// TIA Portal V17 export
// export: Created 2025-03-05T07:59:42.6499915Z, ExportSetting WithDefaults, DisplayName Totally Integrated Automation Portal, DisplayVersion V17 Update 8, DisplayName TIA Portal Openness, DisplayVersion V17 Update 8, DisplayName TIA Portal Version Control Interface, DisplayVersion V17, DisplayName SINAMICS Startdrive Advanced, DisplayVersion V17 SP2, DisplayName SINAMICS Startdrive G110M, G120, G120C, G120D, G120P, G115D, DisplayVersion V17 SP2, DisplayName SINAMICS Startdrive G130, G150, S120, S150, SINAMICS MV, S210, DisplayVersion V17 SP2, DisplayName STEP 7 Professional, DisplayVersion V17 Update 8, DisplayName SINUMERIK ONE STEP 7 Toolbox, DisplayVersion V17 Update 12, DisplayName SINUMERIK 840D sl STEP 7 Toolbox, DisplayVersion V17 Update 12, DisplayName STEP 7 Safety, DisplayVersion V17 Update 6, DisplayName WinCC Advanced, DisplayVersion V17 Update 8
FUNCTION "FC361_NCK_M_CH5_UNIT_2_STA_2" : Void   // FC361, LAD
TITLE = Channel 1 data
{ S7_Optimized_Access := 'FALSE' }
AUTHOR : ETXETAR
VERSION : 1.0
// stored: AutoNumber false, IsIECCheckEnabled false, SetENOAutomatically false, UDAEnableTagReadback false
BEGIN

REGION Network 1: ACKNOWLEDGE M700-FIXTURE 4 CLAMP SEQUENCE (READ-IN DISABLE) / ACKNOWLEDGE M100-CLAMP SEQUENCE FIXTURE 1
   // NOTE: WHEN THERE IS NOT INDEXING TABLE AVAILABLE IN THE MACHINE DELETE 
   // DB2171.DBX5.0 AND DB2171.DBX2.0
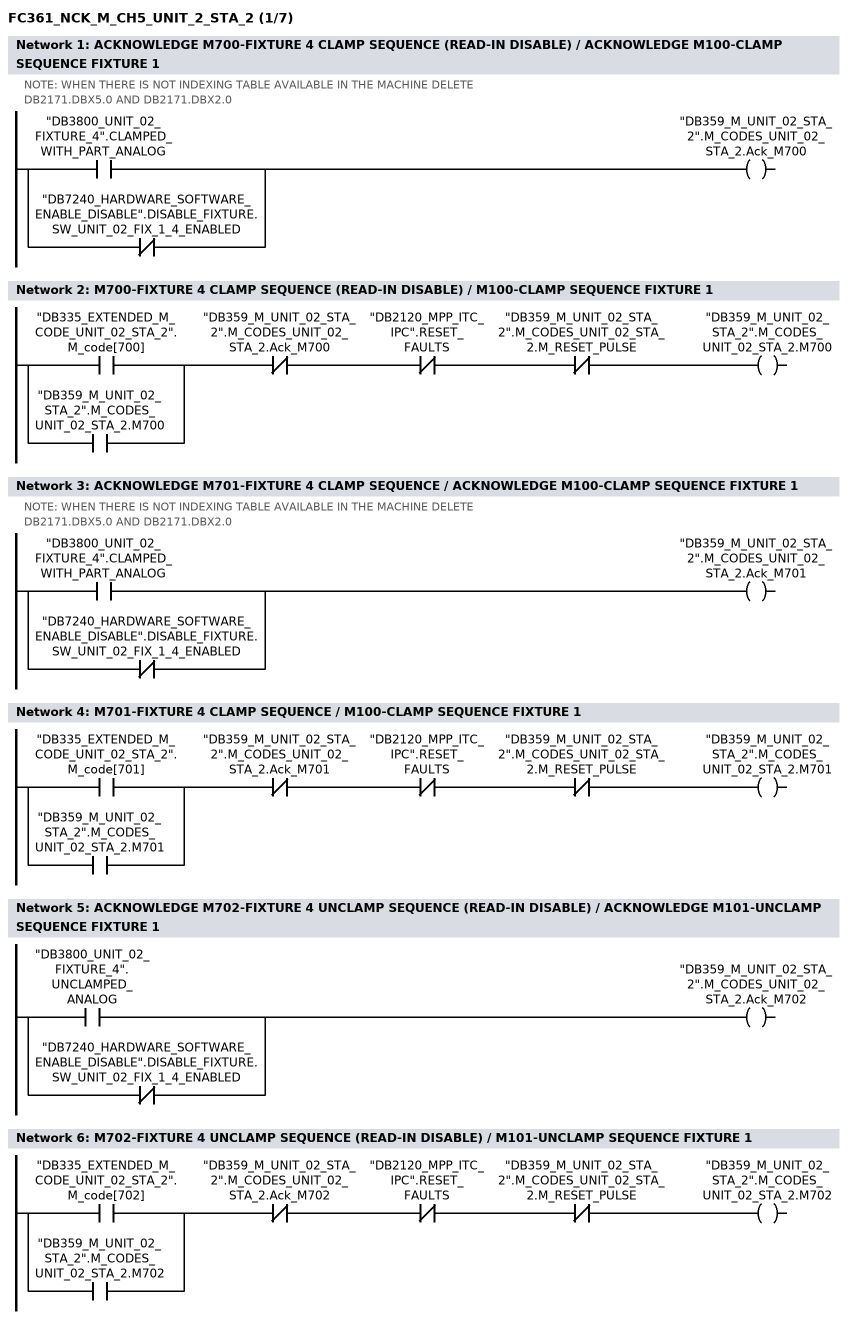
   RUNG wire#powerrail
      Contact( "DB3800_UNIT_02_FIXTURE_4".CLAMPED_WITH_PART_ANALOG )
      wire#w1
      Coil( "DB359_M_UNIT_02_STA_2".M_CODES_UNIT_02_STA_2.Ack_M700 )
   END_RUNG
   RUNG wire#powerrail
      I_Contact( "DB7240_HARDWARE_SOFTWARE_ENABLE_DISABLE".DISABLE_FIXTURE.SW_UNIT_02_FIX_1_4_ENABLED )
   END_RUNG wire#w1
   // the same network as SCL:
   "DB359_M_UNIT_02_STA_2".M_CODES_UNIT_02_STA_2.Ack_M700 := "DB3800_UNIT_02_FIXTURE_4".CLAMPED_WITH_PART_ANALOG OR NOT "DB7240_HARDWARE_SOFTWARE_ENABLE_DISABLE".DISABLE_FIXTURE.SW_UNIT_02_FIX_1_4_ENABLED;
END_REGION

REGION Network 2: M700-FIXTURE 4 CLAMP SEQUENCE (READ-IN DISABLE) / M100-CLAMP SEQUENCE FIXTURE 1
   RUNG wire#powerrail
      Contact( "DB335_EXTENDED_M_CODE_UNIT_02_STA_2".M_code[700] )
      wire#w1
      I_Contact( "DB359_M_UNIT_02_STA_2".M_CODES_UNIT_02_STA_2.Ack_M700 )
      I_Contact( "DB2120_MPP_ITC_IPC".RESET_FAULTS )
      I_Contact( "DB359_M_UNIT_02_STA_2".M_CODES_UNIT_02_STA_2.M_RESET_PULSE )
      Coil( "DB359_M_UNIT_02_STA_2".M_CODES_UNIT_02_STA_2.M700 )
   END_RUNG
   RUNG wire#powerrail
      Contact( "DB359_M_UNIT_02_STA_2".M_CODES_UNIT_02_STA_2.M700 )
   END_RUNG wire#w1
   // the same network as SCL:
   "DB359_M_UNIT_02_STA_2".M_CODES_UNIT_02_STA_2.M700 := ("DB335_EXTENDED_M_CODE_UNIT_02_STA_2".M_code[700] OR "DB359_M_UNIT_02_STA_2".M_CODES_UNIT_02_STA_2.M700) AND NOT "DB359_M_UNIT_02_STA_2".M_CODES_UNIT_02_STA_2.Ack_M700 AND NOT "DB2120_MPP_ITC_IPC".RESET_FAULTS AND NOT "DB359_M_UNIT_02_STA_2".M_CODES_UNIT_02_STA_2.M_RESET_PULSE;
END_REGION

REGION Network 3: ACKNOWLEDGE M701-FIXTURE 4 CLAMP SEQUENCE / ACKNOWLEDGE M100-CLAMP SEQUENCE FIXTURE 1
   // NOTE: WHEN THERE IS NOT INDEXING TABLE AVAILABLE IN THE MACHINE DELETE 
   // DB2171.DBX5.0 AND DB2171.DBX2.0
   RUNG wire#powerrail
      Contact( "DB3800_UNIT_02_FIXTURE_4".CLAMPED_WITH_PART_ANALOG )
      wire#w1
      Coil( "DB359_M_UNIT_02_STA_2".M_CODES_UNIT_02_STA_2.Ack_M701 )
   END_RUNG
   RUNG wire#powerrail
      I_Contact( "DB7240_HARDWARE_SOFTWARE_ENABLE_DISABLE".DISABLE_FIXTURE.SW_UNIT_02_FIX_1_4_ENABLED )
   END_RUNG wire#w1
   // the same network as SCL:
   "DB359_M_UNIT_02_STA_2".M_CODES_UNIT_02_STA_2.Ack_M701 := "DB3800_UNIT_02_FIXTURE_4".CLAMPED_WITH_PART_ANALOG OR NOT "DB7240_HARDWARE_SOFTWARE_ENABLE_DISABLE".DISABLE_FIXTURE.SW_UNIT_02_FIX_1_4_ENABLED;
END_REGION

REGION Network 4: M701-FIXTURE 4 CLAMP SEQUENCE / M100-CLAMP SEQUENCE FIXTURE 1
   RUNG wire#powerrail
      Contact( "DB335_EXTENDED_M_CODE_UNIT_02_STA_2".M_code[701] )
      wire#w1
      I_Contact( "DB359_M_UNIT_02_STA_2".M_CODES_UNIT_02_STA_2.Ack_M701 )
      I_Contact( "DB2120_MPP_ITC_IPC".RESET_FAULTS )
      I_Contact( "DB359_M_UNIT_02_STA_2".M_CODES_UNIT_02_STA_2.M_RESET_PULSE )
      Coil( "DB359_M_UNIT_02_STA_2".M_CODES_UNIT_02_STA_2.M701 )
   END_RUNG
   RUNG wire#powerrail
      Contact( "DB359_M_UNIT_02_STA_2".M_CODES_UNIT_02_STA_2.M701 )
   END_RUNG wire#w1
   // the same network as SCL:
   "DB359_M_UNIT_02_STA_2".M_CODES_UNIT_02_STA_2.M701 := ("DB335_EXTENDED_M_CODE_UNIT_02_STA_2".M_code[701] OR "DB359_M_UNIT_02_STA_2".M_CODES_UNIT_02_STA_2.M701) AND NOT "DB359_M_UNIT_02_STA_2".M_CODES_UNIT_02_STA_2.Ack_M701 AND NOT "DB2120_MPP_ITC_IPC".RESET_FAULTS AND NOT "DB359_M_UNIT_02_STA_2".M_CODES_UNIT_02_STA_2.M_RESET_PULSE;
END_REGION

REGION Network 5: ACKNOWLEDGE M702-FIXTURE 4 UNCLAMP SEQUENCE (READ-IN DISABLE) / ACKNOWLEDGE M101-UNCLAMP SEQUENCE FIXTURE 1
   RUNG wire#powerrail
      Contact( "DB3800_UNIT_02_FIXTURE_4".UNCLAMPED_ANALOG )
      wire#w1
      Coil( "DB359_M_UNIT_02_STA_2".M_CODES_UNIT_02_STA_2.Ack_M702 )
   END_RUNG
   RUNG wire#powerrail
      I_Contact( "DB7240_HARDWARE_SOFTWARE_ENABLE_DISABLE".DISABLE_FIXTURE.SW_UNIT_02_FIX_1_4_ENABLED )
   END_RUNG wire#w1
   // the same network as SCL:
   "DB359_M_UNIT_02_STA_2".M_CODES_UNIT_02_STA_2.Ack_M702 := "DB3800_UNIT_02_FIXTURE_4".UNCLAMPED_ANALOG OR NOT "DB7240_HARDWARE_SOFTWARE_ENABLE_DISABLE".DISABLE_FIXTURE.SW_UNIT_02_FIX_1_4_ENABLED;
END_REGION

REGION Network 6: M702-FIXTURE 4 UNCLAMP SEQUENCE (READ-IN DISABLE) / M101-UNCLAMP SEQUENCE FIXTURE 1
   RUNG wire#powerrail
      Contact( "DB335_EXTENDED_M_CODE_UNIT_02_STA_2".M_code[702] )
      wire#w1
      I_Contact( "DB359_M_UNIT_02_STA_2".M_CODES_UNIT_02_STA_2.Ack_M702 )
      I_Contact( "DB2120_MPP_ITC_IPC".RESET_FAULTS )
      I_Contact( "DB359_M_UNIT_02_STA_2".M_CODES_UNIT_02_STA_2.M_RESET_PULSE )
      Coil( "DB359_M_UNIT_02_STA_2".M_CODES_UNIT_02_STA_2.M702 )
   END_RUNG
   RUNG wire#powerrail
      Contact( "DB359_M_UNIT_02_STA_2".M_CODES_UNIT_02_STA_2.M702 )
   END_RUNG wire#w1
   // the same network as SCL:
   "DB359_M_UNIT_02_STA_2".M_CODES_UNIT_02_STA_2.M702 := ("DB335_EXTENDED_M_CODE_UNIT_02_STA_2".M_code[702] OR "DB359_M_UNIT_02_STA_2".M_CODES_UNIT_02_STA_2.M702) AND NOT "DB359_M_UNIT_02_STA_2".M_CODES_UNIT_02_STA_2.Ack_M702 AND NOT "DB2120_MPP_ITC_IPC".RESET_FAULTS AND NOT "DB359_M_UNIT_02_STA_2".M_CODES_UNIT_02_STA_2.M_RESET_PULSE;
END_REGION

REGION Network 7: ACKNOWLEDGE M703-FIXTURE 4 UNCLAMP SEQUENCE / ACKNOWLEDGE M101-UNCLAMP SEQUENCE FIXTURE 1
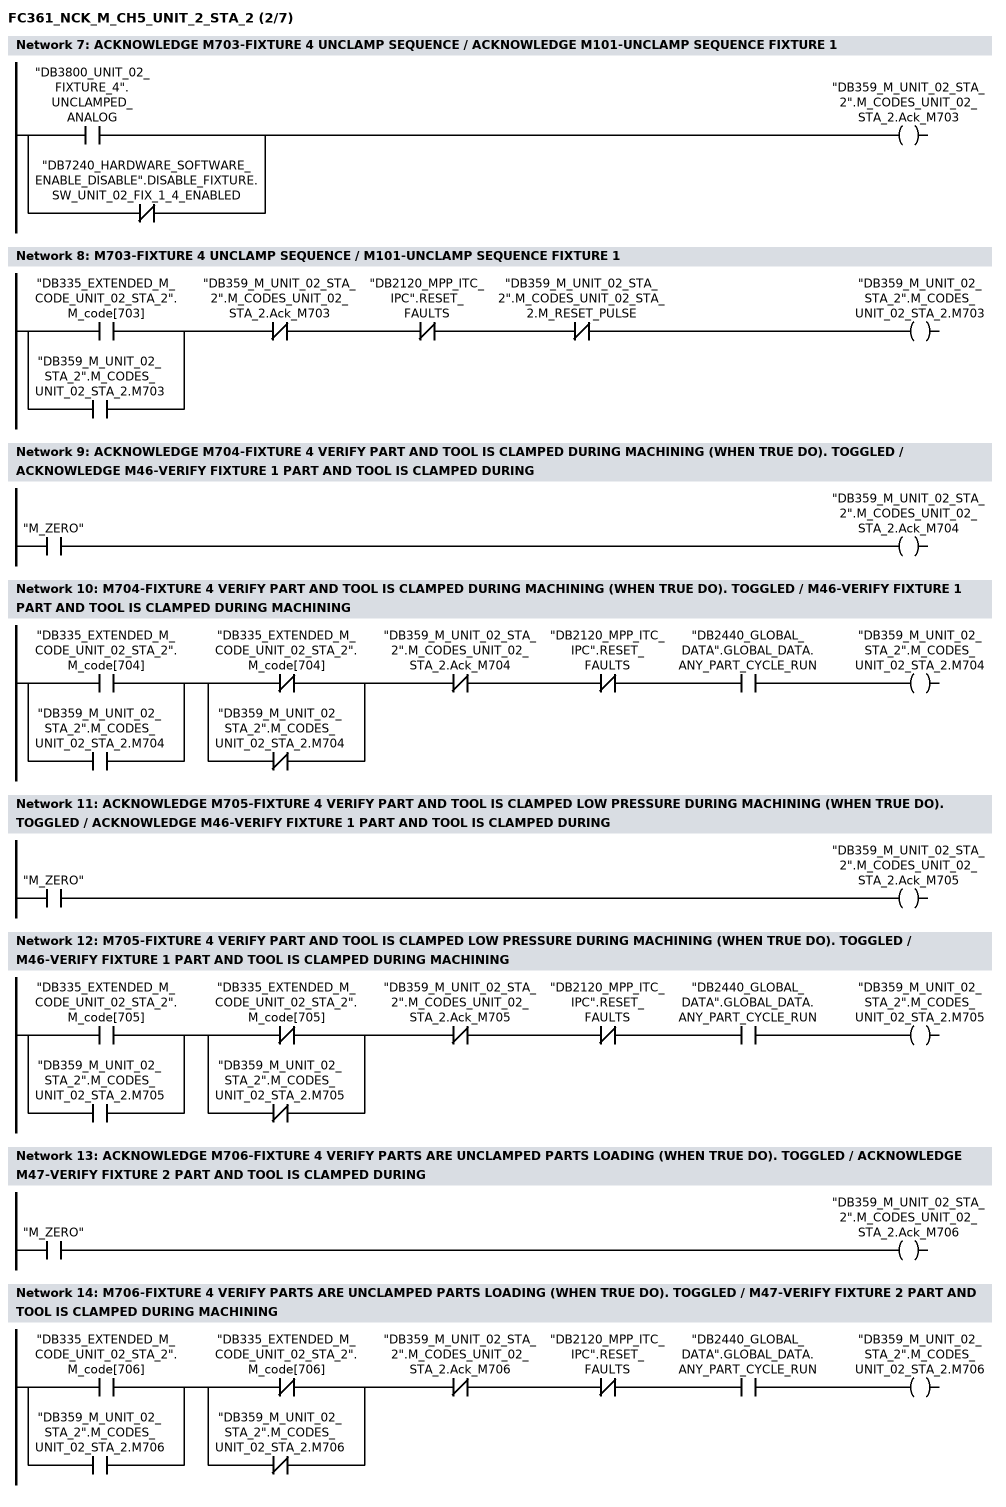
   RUNG wire#powerrail
      Contact( "DB3800_UNIT_02_FIXTURE_4".UNCLAMPED_ANALOG )
      wire#w1
      Coil( "DB359_M_UNIT_02_STA_2".M_CODES_UNIT_02_STA_2.Ack_M703 )
   END_RUNG
   RUNG wire#powerrail
      I_Contact( "DB7240_HARDWARE_SOFTWARE_ENABLE_DISABLE".DISABLE_FIXTURE.SW_UNIT_02_FIX_1_4_ENABLED )
   END_RUNG wire#w1
   // the same network as SCL:
   "DB359_M_UNIT_02_STA_2".M_CODES_UNIT_02_STA_2.Ack_M703 := "DB3800_UNIT_02_FIXTURE_4".UNCLAMPED_ANALOG OR NOT "DB7240_HARDWARE_SOFTWARE_ENABLE_DISABLE".DISABLE_FIXTURE.SW_UNIT_02_FIX_1_4_ENABLED;
END_REGION

REGION Network 8: M703-FIXTURE 4 UNCLAMP SEQUENCE / M101-UNCLAMP SEQUENCE FIXTURE 1
   RUNG wire#powerrail
      Contact( "DB335_EXTENDED_M_CODE_UNIT_02_STA_2".M_code[703] )
      wire#w1
      I_Contact( "DB359_M_UNIT_02_STA_2".M_CODES_UNIT_02_STA_2.Ack_M703 )
      I_Contact( "DB2120_MPP_ITC_IPC".RESET_FAULTS )
      I_Contact( "DB359_M_UNIT_02_STA_2".M_CODES_UNIT_02_STA_2.M_RESET_PULSE )
      Coil( "DB359_M_UNIT_02_STA_2".M_CODES_UNIT_02_STA_2.M703 )
   END_RUNG
   RUNG wire#powerrail
      Contact( "DB359_M_UNIT_02_STA_2".M_CODES_UNIT_02_STA_2.M703 )
   END_RUNG wire#w1
   // the same network as SCL:
   "DB359_M_UNIT_02_STA_2".M_CODES_UNIT_02_STA_2.M703 := ("DB335_EXTENDED_M_CODE_UNIT_02_STA_2".M_code[703] OR "DB359_M_UNIT_02_STA_2".M_CODES_UNIT_02_STA_2.M703) AND NOT "DB359_M_UNIT_02_STA_2".M_CODES_UNIT_02_STA_2.Ack_M703 AND NOT "DB2120_MPP_ITC_IPC".RESET_FAULTS AND NOT "DB359_M_UNIT_02_STA_2".M_CODES_UNIT_02_STA_2.M_RESET_PULSE;
END_REGION

REGION Network 9: ACKNOWLEDGE M704-FIXTURE 4 VERIFY PART AND TOOL IS CLAMPED DURING MACHINING (WHEN TRUE DO). TOGGLED / ACKNOWLEDGE M46-VERIFY FIXTURE 1 PART AND TOOL IS CLAMPED DURING
   RUNG wire#powerrail
      Contact( "M_ZERO" )
      Coil( "DB359_M_UNIT_02_STA_2".M_CODES_UNIT_02_STA_2.Ack_M704 )
   END_RUNG
   // the same network as SCL:
   "DB359_M_UNIT_02_STA_2".M_CODES_UNIT_02_STA_2.Ack_M704 := "M_ZERO";
END_REGION

REGION Network 10: M704-FIXTURE 4 VERIFY PART AND TOOL IS CLAMPED DURING MACHINING (WHEN TRUE DO). TOGGLED / M46-VERIFY FIXTURE 1 PART AND TOOL IS CLAMPED DURING MACHINING
   RUNG wire#powerrail
      Contact( "DB335_EXTENDED_M_CODE_UNIT_02_STA_2".M_code[704] )
      wire#w1
      I_Contact( "DB335_EXTENDED_M_CODE_UNIT_02_STA_2".M_code[704] )
      wire#w2
      I_Contact( "DB359_M_UNIT_02_STA_2".M_CODES_UNIT_02_STA_2.Ack_M704 )
      I_Contact( "DB2120_MPP_ITC_IPC".RESET_FAULTS )
      Contact( "DB2440_GLOBAL_DATA".GLOBAL_DATA.ANY_PART_CYCLE_RUN )
      Coil( "DB359_M_UNIT_02_STA_2".M_CODES_UNIT_02_STA_2.M704 )
   END_RUNG
   RUNG wire#powerrail
      Contact( "DB359_M_UNIT_02_STA_2".M_CODES_UNIT_02_STA_2.M704 )
   END_RUNG wire#w1
   RUNG wire#w1
      I_Contact( "DB359_M_UNIT_02_STA_2".M_CODES_UNIT_02_STA_2.M704 )
   END_RUNG wire#w2
   // the same network as SCL:
   "DB359_M_UNIT_02_STA_2".M_CODES_UNIT_02_STA_2.M704 := ("DB335_EXTENDED_M_CODE_UNIT_02_STA_2".M_code[704] OR "DB359_M_UNIT_02_STA_2".M_CODES_UNIT_02_STA_2.M704) AND (NOT "DB335_EXTENDED_M_CODE_UNIT_02_STA_2".M_code[704] OR NOT "DB359_M_UNIT_02_STA_2".M_CODES_UNIT_02_STA_2.M704) AND NOT "DB359_M_UNIT_02_STA_2".M_CODES_UNIT_02_STA_2.Ack_M704 AND NOT "DB2120_MPP_ITC_IPC".RESET_FAULTS AND "DB2440_GLOBAL_DATA".GLOBAL_DATA.ANY_PART_CYCLE_RUN;
END_REGION

REGION Network 11: ACKNOWLEDGE M705-FIXTURE 4 VERIFY PART AND TOOL IS CLAMPED LOW PRESSURE DURING MACHINING (WHEN TRUE DO). TOGGLED / ACKNOWLEDGE M46-VERIFY FIXTURE 1 PART AND TOOL IS CLAMPED DURING
   RUNG wire#powerrail
      Contact( "M_ZERO" )
      Coil( "DB359_M_UNIT_02_STA_2".M_CODES_UNIT_02_STA_2.Ack_M705 )
   END_RUNG
   // the same network as SCL:
   "DB359_M_UNIT_02_STA_2".M_CODES_UNIT_02_STA_2.Ack_M705 := "M_ZERO";
END_REGION

REGION Network 12: M705-FIXTURE 4 VERIFY PART AND TOOL IS CLAMPED LOW PRESSURE DURING MACHINING (WHEN TRUE DO). TOGGLED / M46-VERIFY FIXTURE 1 PART AND TOOL IS CLAMPED DURING MACHINING
   RUNG wire#powerrail
      Contact( "DB335_EXTENDED_M_CODE_UNIT_02_STA_2".M_code[705] )
      wire#w1
      I_Contact( "DB335_EXTENDED_M_CODE_UNIT_02_STA_2".M_code[705] )
      wire#w2
      I_Contact( "DB359_M_UNIT_02_STA_2".M_CODES_UNIT_02_STA_2.Ack_M705 )
      I_Contact( "DB2120_MPP_ITC_IPC".RESET_FAULTS )
      Contact( "DB2440_GLOBAL_DATA".GLOBAL_DATA.ANY_PART_CYCLE_RUN )
      Coil( "DB359_M_UNIT_02_STA_2".M_CODES_UNIT_02_STA_2.M705 )
   END_RUNG
   RUNG wire#powerrail
      Contact( "DB359_M_UNIT_02_STA_2".M_CODES_UNIT_02_STA_2.M705 )
   END_RUNG wire#w1
   RUNG wire#w1
      I_Contact( "DB359_M_UNIT_02_STA_2".M_CODES_UNIT_02_STA_2.M705 )
   END_RUNG wire#w2
   // the same network as SCL:
   "DB359_M_UNIT_02_STA_2".M_CODES_UNIT_02_STA_2.M705 := ("DB335_EXTENDED_M_CODE_UNIT_02_STA_2".M_code[705] OR "DB359_M_UNIT_02_STA_2".M_CODES_UNIT_02_STA_2.M705) AND (NOT "DB335_EXTENDED_M_CODE_UNIT_02_STA_2".M_code[705] OR NOT "DB359_M_UNIT_02_STA_2".M_CODES_UNIT_02_STA_2.M705) AND NOT "DB359_M_UNIT_02_STA_2".M_CODES_UNIT_02_STA_2.Ack_M705 AND NOT "DB2120_MPP_ITC_IPC".RESET_FAULTS AND "DB2440_GLOBAL_DATA".GLOBAL_DATA.ANY_PART_CYCLE_RUN;
END_REGION

REGION Network 13: ACKNOWLEDGE M706-FIXTURE 4 VERIFY PARTS ARE UNCLAMPED PARTS LOADING (WHEN TRUE DO). TOGGLED / ACKNOWLEDGE M47-VERIFY FIXTURE 2 PART AND TOOL IS CLAMPED DURING
   RUNG wire#powerrail
      Contact( "M_ZERO" )
      Coil( "DB359_M_UNIT_02_STA_2".M_CODES_UNIT_02_STA_2.Ack_M706 )
   END_RUNG
   // the same network as SCL:
   "DB359_M_UNIT_02_STA_2".M_CODES_UNIT_02_STA_2.Ack_M706 := "M_ZERO";
END_REGION

REGION Network 14: M706-FIXTURE 4 VERIFY PARTS ARE UNCLAMPED PARTS LOADING (WHEN TRUE DO). TOGGLED / M47-VERIFY FIXTURE 2 PART AND TOOL IS CLAMPED DURING MACHINING
   RUNG wire#powerrail
      Contact( "DB335_EXTENDED_M_CODE_UNIT_02_STA_2".M_code[706] )
      wire#w1
      I_Contact( "DB335_EXTENDED_M_CODE_UNIT_02_STA_2".M_code[706] )
      wire#w2
      I_Contact( "DB359_M_UNIT_02_STA_2".M_CODES_UNIT_02_STA_2.Ack_M706 )
      I_Contact( "DB2120_MPP_ITC_IPC".RESET_FAULTS )
      Contact( "DB2440_GLOBAL_DATA".GLOBAL_DATA.ANY_PART_CYCLE_RUN )
      Coil( "DB359_M_UNIT_02_STA_2".M_CODES_UNIT_02_STA_2.M706 )
   END_RUNG
   RUNG wire#powerrail
      Contact( "DB359_M_UNIT_02_STA_2".M_CODES_UNIT_02_STA_2.M706 )
   END_RUNG wire#w1
   RUNG wire#w1
      I_Contact( "DB359_M_UNIT_02_STA_2".M_CODES_UNIT_02_STA_2.M706 )
   END_RUNG wire#w2
   // the same network as SCL:
   "DB359_M_UNIT_02_STA_2".M_CODES_UNIT_02_STA_2.M706 := ("DB335_EXTENDED_M_CODE_UNIT_02_STA_2".M_code[706] OR "DB359_M_UNIT_02_STA_2".M_CODES_UNIT_02_STA_2.M706) AND (NOT "DB335_EXTENDED_M_CODE_UNIT_02_STA_2".M_code[706] OR NOT "DB359_M_UNIT_02_STA_2".M_CODES_UNIT_02_STA_2.M706) AND NOT "DB359_M_UNIT_02_STA_2".M_CODES_UNIT_02_STA_2.Ack_M706 AND NOT "DB2120_MPP_ITC_IPC".RESET_FAULTS AND "DB2440_GLOBAL_DATA".GLOBAL_DATA.ANY_PART_CYCLE_RUN;
END_REGION

REGION Network 15: ACKNOWLEDGE M707-FIXTURE 4 VERIFY FIXTURE REMAINS CLAMPED
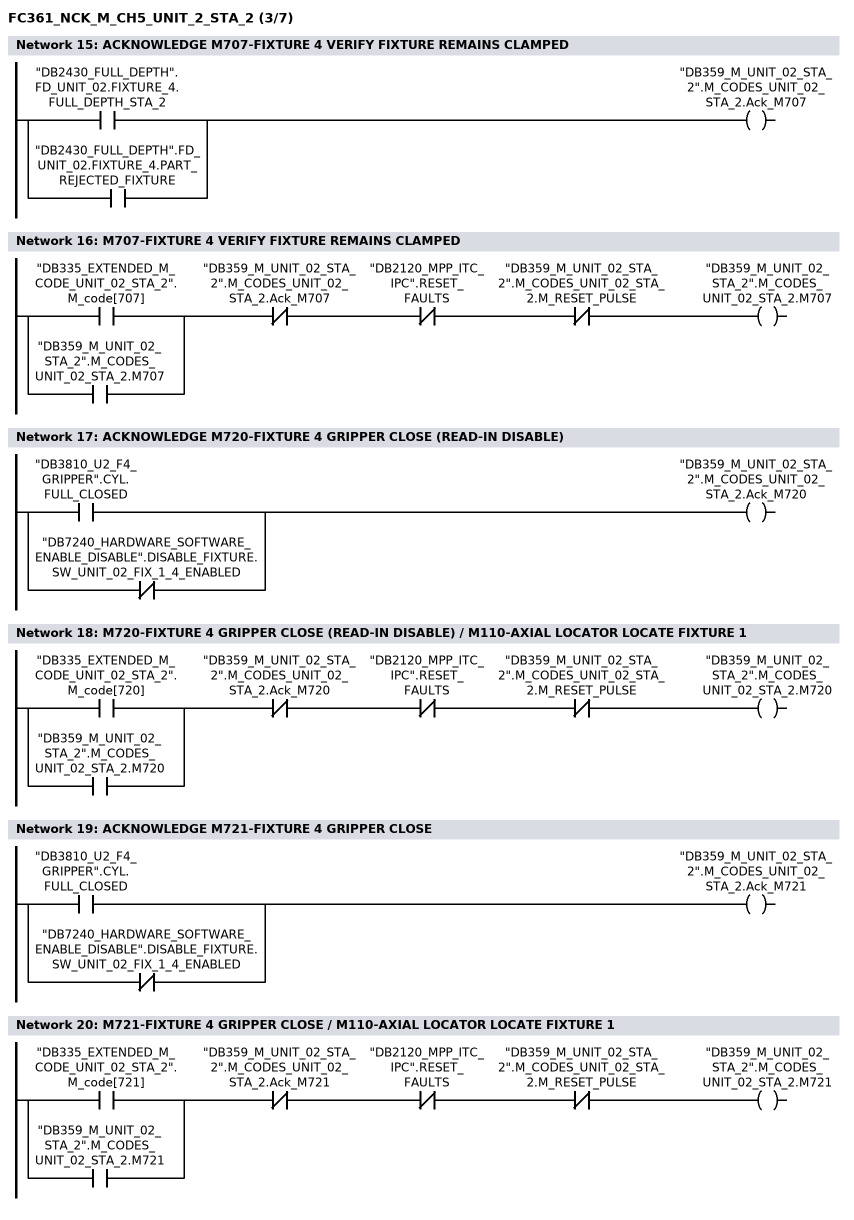
   RUNG wire#powerrail
      Contact( "DB2430_FULL_DEPTH".FD_UNIT_02.FIXTURE_4.FULL_DEPTH_STA_2 )
      wire#w1
      Coil( "DB359_M_UNIT_02_STA_2".M_CODES_UNIT_02_STA_2.Ack_M707 )
   END_RUNG
   RUNG wire#powerrail
      Contact( "DB2430_FULL_DEPTH".FD_UNIT_02.FIXTURE_4.PART_REJECTED_FIXTURE )
   END_RUNG wire#w1
   // the same network as SCL:
   "DB359_M_UNIT_02_STA_2".M_CODES_UNIT_02_STA_2.Ack_M707 := "DB2430_FULL_DEPTH".FD_UNIT_02.FIXTURE_4.FULL_DEPTH_STA_2 OR "DB2430_FULL_DEPTH".FD_UNIT_02.FIXTURE_4.PART_REJECTED_FIXTURE;
END_REGION

REGION Network 16: M707-FIXTURE 4 VERIFY FIXTURE REMAINS CLAMPED
   RUNG wire#powerrail
      Contact( "DB335_EXTENDED_M_CODE_UNIT_02_STA_2".M_code[707] )
      wire#w1
      I_Contact( "DB359_M_UNIT_02_STA_2".M_CODES_UNIT_02_STA_2.Ack_M707 )
      I_Contact( "DB2120_MPP_ITC_IPC".RESET_FAULTS )
      I_Contact( "DB359_M_UNIT_02_STA_2".M_CODES_UNIT_02_STA_2.M_RESET_PULSE )
      Coil( "DB359_M_UNIT_02_STA_2".M_CODES_UNIT_02_STA_2.M707 )
   END_RUNG
   RUNG wire#powerrail
      Contact( "DB359_M_UNIT_02_STA_2".M_CODES_UNIT_02_STA_2.M707 )
   END_RUNG wire#w1
   // the same network as SCL:
   "DB359_M_UNIT_02_STA_2".M_CODES_UNIT_02_STA_2.M707 := ("DB335_EXTENDED_M_CODE_UNIT_02_STA_2".M_code[707] OR "DB359_M_UNIT_02_STA_2".M_CODES_UNIT_02_STA_2.M707) AND NOT "DB359_M_UNIT_02_STA_2".M_CODES_UNIT_02_STA_2.Ack_M707 AND NOT "DB2120_MPP_ITC_IPC".RESET_FAULTS AND NOT "DB359_M_UNIT_02_STA_2".M_CODES_UNIT_02_STA_2.M_RESET_PULSE;
END_REGION

REGION Network 17: ACKNOWLEDGE M720-FIXTURE 4 GRIPPER CLOSE (READ-IN DISABLE)
   RUNG wire#powerrail
      Contact( "DB3810_U2_F4_GRIPPER".CYL.FULL_CLOSED )
      wire#w1
      Coil( "DB359_M_UNIT_02_STA_2".M_CODES_UNIT_02_STA_2.Ack_M720 )
   END_RUNG
   RUNG wire#powerrail
      I_Contact( "DB7240_HARDWARE_SOFTWARE_ENABLE_DISABLE".DISABLE_FIXTURE.SW_UNIT_02_FIX_1_4_ENABLED )
   END_RUNG wire#w1
   // the same network as SCL:
   "DB359_M_UNIT_02_STA_2".M_CODES_UNIT_02_STA_2.Ack_M720 := "DB3810_U2_F4_GRIPPER".CYL.FULL_CLOSED OR NOT "DB7240_HARDWARE_SOFTWARE_ENABLE_DISABLE".DISABLE_FIXTURE.SW_UNIT_02_FIX_1_4_ENABLED;
END_REGION

REGION Network 18: M720-FIXTURE 4 GRIPPER CLOSE (READ-IN DISABLE) / M110-AXIAL LOCATOR LOCATE FIXTURE 1
   RUNG wire#powerrail
      Contact( "DB335_EXTENDED_M_CODE_UNIT_02_STA_2".M_code[720] )
      wire#w1
      I_Contact( "DB359_M_UNIT_02_STA_2".M_CODES_UNIT_02_STA_2.Ack_M720 )
      I_Contact( "DB2120_MPP_ITC_IPC".RESET_FAULTS )
      I_Contact( "DB359_M_UNIT_02_STA_2".M_CODES_UNIT_02_STA_2.M_RESET_PULSE )
      Coil( "DB359_M_UNIT_02_STA_2".M_CODES_UNIT_02_STA_2.M720 )
   END_RUNG
   RUNG wire#powerrail
      Contact( "DB359_M_UNIT_02_STA_2".M_CODES_UNIT_02_STA_2.M720 )
   END_RUNG wire#w1
   // the same network as SCL:
   "DB359_M_UNIT_02_STA_2".M_CODES_UNIT_02_STA_2.M720 := ("DB335_EXTENDED_M_CODE_UNIT_02_STA_2".M_code[720] OR "DB359_M_UNIT_02_STA_2".M_CODES_UNIT_02_STA_2.M720) AND NOT "DB359_M_UNIT_02_STA_2".M_CODES_UNIT_02_STA_2.Ack_M720 AND NOT "DB2120_MPP_ITC_IPC".RESET_FAULTS AND NOT "DB359_M_UNIT_02_STA_2".M_CODES_UNIT_02_STA_2.M_RESET_PULSE;
END_REGION

REGION Network 19: ACKNOWLEDGE M721-FIXTURE 4 GRIPPER CLOSE
   RUNG wire#powerrail
      Contact( "DB3810_U2_F4_GRIPPER".CYL.FULL_CLOSED )
      wire#w1
      Coil( "DB359_M_UNIT_02_STA_2".M_CODES_UNIT_02_STA_2.Ack_M721 )
   END_RUNG
   RUNG wire#powerrail
      I_Contact( "DB7240_HARDWARE_SOFTWARE_ENABLE_DISABLE".DISABLE_FIXTURE.SW_UNIT_02_FIX_1_4_ENABLED )
   END_RUNG wire#w1
   // the same network as SCL:
   "DB359_M_UNIT_02_STA_2".M_CODES_UNIT_02_STA_2.Ack_M721 := "DB3810_U2_F4_GRIPPER".CYL.FULL_CLOSED OR NOT "DB7240_HARDWARE_SOFTWARE_ENABLE_DISABLE".DISABLE_FIXTURE.SW_UNIT_02_FIX_1_4_ENABLED;
END_REGION

REGION Network 20: M721-FIXTURE 4 GRIPPER CLOSE / M110-AXIAL LOCATOR LOCATE FIXTURE 1
   RUNG wire#powerrail
      Contact( "DB335_EXTENDED_M_CODE_UNIT_02_STA_2".M_code[721] )
      wire#w1
      I_Contact( "DB359_M_UNIT_02_STA_2".M_CODES_UNIT_02_STA_2.Ack_M721 )
      I_Contact( "DB2120_MPP_ITC_IPC".RESET_FAULTS )
      I_Contact( "DB359_M_UNIT_02_STA_2".M_CODES_UNIT_02_STA_2.M_RESET_PULSE )
      Coil( "DB359_M_UNIT_02_STA_2".M_CODES_UNIT_02_STA_2.M721 )
   END_RUNG
   RUNG wire#powerrail
      Contact( "DB359_M_UNIT_02_STA_2".M_CODES_UNIT_02_STA_2.M721 )
   END_RUNG wire#w1
   // the same network as SCL:
   "DB359_M_UNIT_02_STA_2".M_CODES_UNIT_02_STA_2.M721 := ("DB335_EXTENDED_M_CODE_UNIT_02_STA_2".M_code[721] OR "DB359_M_UNIT_02_STA_2".M_CODES_UNIT_02_STA_2.M721) AND NOT "DB359_M_UNIT_02_STA_2".M_CODES_UNIT_02_STA_2.Ack_M721 AND NOT "DB2120_MPP_ITC_IPC".RESET_FAULTS AND NOT "DB359_M_UNIT_02_STA_2".M_CODES_UNIT_02_STA_2.M_RESET_PULSE;
END_REGION

REGION Network 21: ACKNOWLEDGE M722-FIXTURE 4 GRIPPER RETURN (READ-IN DISABLE) / ACKNOWLEDGE M111-AXIAL LOCATOR RETURN FIXTURE 1
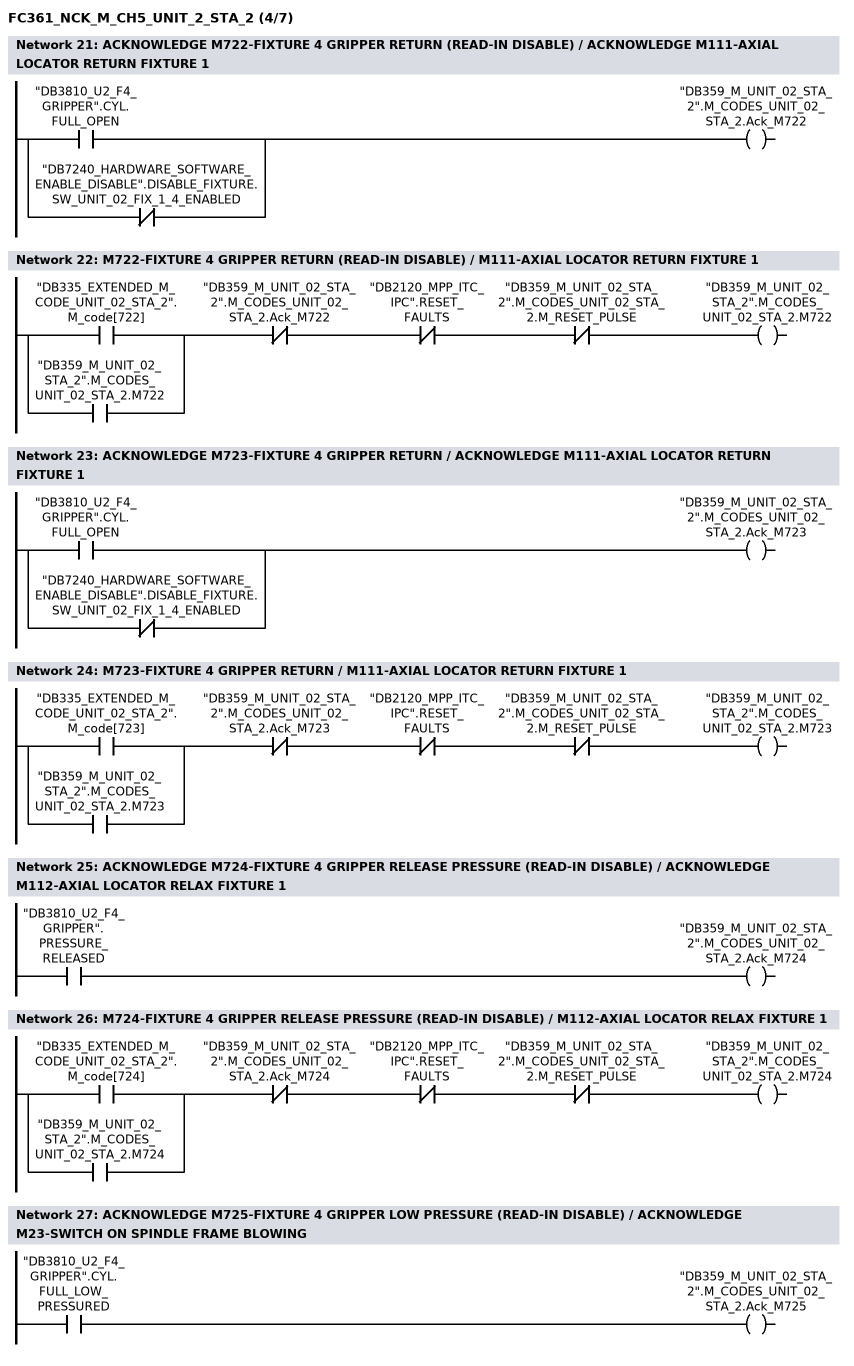
   RUNG wire#powerrail
      Contact( "DB3810_U2_F4_GRIPPER".CYL.FULL_OPEN )
      wire#w1
      Coil( "DB359_M_UNIT_02_STA_2".M_CODES_UNIT_02_STA_2.Ack_M722 )
   END_RUNG
   RUNG wire#powerrail
      I_Contact( "DB7240_HARDWARE_SOFTWARE_ENABLE_DISABLE".DISABLE_FIXTURE.SW_UNIT_02_FIX_1_4_ENABLED )
   END_RUNG wire#w1
   // the same network as SCL:
   "DB359_M_UNIT_02_STA_2".M_CODES_UNIT_02_STA_2.Ack_M722 := "DB3810_U2_F4_GRIPPER".CYL.FULL_OPEN OR NOT "DB7240_HARDWARE_SOFTWARE_ENABLE_DISABLE".DISABLE_FIXTURE.SW_UNIT_02_FIX_1_4_ENABLED;
END_REGION

REGION Network 22: M722-FIXTURE 4 GRIPPER RETURN (READ-IN DISABLE) / M111-AXIAL LOCATOR RETURN FIXTURE 1
   RUNG wire#powerrail
      Contact( "DB335_EXTENDED_M_CODE_UNIT_02_STA_2".M_code[722] )
      wire#w1
      I_Contact( "DB359_M_UNIT_02_STA_2".M_CODES_UNIT_02_STA_2.Ack_M722 )
      I_Contact( "DB2120_MPP_ITC_IPC".RESET_FAULTS )
      I_Contact( "DB359_M_UNIT_02_STA_2".M_CODES_UNIT_02_STA_2.M_RESET_PULSE )
      Coil( "DB359_M_UNIT_02_STA_2".M_CODES_UNIT_02_STA_2.M722 )
   END_RUNG
   RUNG wire#powerrail
      Contact( "DB359_M_UNIT_02_STA_2".M_CODES_UNIT_02_STA_2.M722 )
   END_RUNG wire#w1
   // the same network as SCL:
   "DB359_M_UNIT_02_STA_2".M_CODES_UNIT_02_STA_2.M722 := ("DB335_EXTENDED_M_CODE_UNIT_02_STA_2".M_code[722] OR "DB359_M_UNIT_02_STA_2".M_CODES_UNIT_02_STA_2.M722) AND NOT "DB359_M_UNIT_02_STA_2".M_CODES_UNIT_02_STA_2.Ack_M722 AND NOT "DB2120_MPP_ITC_IPC".RESET_FAULTS AND NOT "DB359_M_UNIT_02_STA_2".M_CODES_UNIT_02_STA_2.M_RESET_PULSE;
END_REGION

REGION Network 23: ACKNOWLEDGE M723-FIXTURE 4 GRIPPER RETURN / ACKNOWLEDGE M111-AXIAL LOCATOR RETURN FIXTURE 1
   RUNG wire#powerrail
      Contact( "DB3810_U2_F4_GRIPPER".CYL.FULL_OPEN )
      wire#w1
      Coil( "DB359_M_UNIT_02_STA_2".M_CODES_UNIT_02_STA_2.Ack_M723 )
   END_RUNG
   RUNG wire#powerrail
      I_Contact( "DB7240_HARDWARE_SOFTWARE_ENABLE_DISABLE".DISABLE_FIXTURE.SW_UNIT_02_FIX_1_4_ENABLED )
   END_RUNG wire#w1
   // the same network as SCL:
   "DB359_M_UNIT_02_STA_2".M_CODES_UNIT_02_STA_2.Ack_M723 := "DB3810_U2_F4_GRIPPER".CYL.FULL_OPEN OR NOT "DB7240_HARDWARE_SOFTWARE_ENABLE_DISABLE".DISABLE_FIXTURE.SW_UNIT_02_FIX_1_4_ENABLED;
END_REGION

REGION Network 24: M723-FIXTURE 4 GRIPPER RETURN / M111-AXIAL LOCATOR RETURN FIXTURE 1
   RUNG wire#powerrail
      Contact( "DB335_EXTENDED_M_CODE_UNIT_02_STA_2".M_code[723] )
      wire#w1
      I_Contact( "DB359_M_UNIT_02_STA_2".M_CODES_UNIT_02_STA_2.Ack_M723 )
      I_Contact( "DB2120_MPP_ITC_IPC".RESET_FAULTS )
      I_Contact( "DB359_M_UNIT_02_STA_2".M_CODES_UNIT_02_STA_2.M_RESET_PULSE )
      Coil( "DB359_M_UNIT_02_STA_2".M_CODES_UNIT_02_STA_2.M723 )
   END_RUNG
   RUNG wire#powerrail
      Contact( "DB359_M_UNIT_02_STA_2".M_CODES_UNIT_02_STA_2.M723 )
   END_RUNG wire#w1
   // the same network as SCL:
   "DB359_M_UNIT_02_STA_2".M_CODES_UNIT_02_STA_2.M723 := ("DB335_EXTENDED_M_CODE_UNIT_02_STA_2".M_code[723] OR "DB359_M_UNIT_02_STA_2".M_CODES_UNIT_02_STA_2.M723) AND NOT "DB359_M_UNIT_02_STA_2".M_CODES_UNIT_02_STA_2.Ack_M723 AND NOT "DB2120_MPP_ITC_IPC".RESET_FAULTS AND NOT "DB359_M_UNIT_02_STA_2".M_CODES_UNIT_02_STA_2.M_RESET_PULSE;
END_REGION

REGION Network 25: ACKNOWLEDGE M724-FIXTURE 4 GRIPPER RELEASE PRESSURE (READ-IN DISABLE) / ACKNOWLEDGE M112-AXIAL LOCATOR RELAX FIXTURE 1
   RUNG wire#powerrail
      Contact( "DB3810_U2_F4_GRIPPER".PRESSURE_RELEASED )
      Coil( "DB359_M_UNIT_02_STA_2".M_CODES_UNIT_02_STA_2.Ack_M724 )
   END_RUNG
   // the same network as SCL:
   "DB359_M_UNIT_02_STA_2".M_CODES_UNIT_02_STA_2.Ack_M724 := "DB3810_U2_F4_GRIPPER".PRESSURE_RELEASED;
END_REGION

REGION Network 26: M724-FIXTURE 4 GRIPPER RELEASE PRESSURE (READ-IN DISABLE) / M112-AXIAL LOCATOR RELAX FIXTURE 1
   RUNG wire#powerrail
      Contact( "DB335_EXTENDED_M_CODE_UNIT_02_STA_2".M_code[724] )
      wire#w1
      I_Contact( "DB359_M_UNIT_02_STA_2".M_CODES_UNIT_02_STA_2.Ack_M724 )
      I_Contact( "DB2120_MPP_ITC_IPC".RESET_FAULTS )
      I_Contact( "DB359_M_UNIT_02_STA_2".M_CODES_UNIT_02_STA_2.M_RESET_PULSE )
      Coil( "DB359_M_UNIT_02_STA_2".M_CODES_UNIT_02_STA_2.M724 )
   END_RUNG
   RUNG wire#powerrail
      Contact( "DB359_M_UNIT_02_STA_2".M_CODES_UNIT_02_STA_2.M724 )
   END_RUNG wire#w1
   // the same network as SCL:
   "DB359_M_UNIT_02_STA_2".M_CODES_UNIT_02_STA_2.M724 := ("DB335_EXTENDED_M_CODE_UNIT_02_STA_2".M_code[724] OR "DB359_M_UNIT_02_STA_2".M_CODES_UNIT_02_STA_2.M724) AND NOT "DB359_M_UNIT_02_STA_2".M_CODES_UNIT_02_STA_2.Ack_M724 AND NOT "DB2120_MPP_ITC_IPC".RESET_FAULTS AND NOT "DB359_M_UNIT_02_STA_2".M_CODES_UNIT_02_STA_2.M_RESET_PULSE;
END_REGION

REGION Network 27: ACKNOWLEDGE M725-FIXTURE 4 GRIPPER LOW PRESSURE (READ-IN DISABLE) / ACKNOWLEDGE M23-SWITCH ON SPINDLE FRAME BLOWING
   RUNG wire#powerrail
      Contact( "DB3810_U2_F4_GRIPPER".CYL.FULL_LOW_PRESSURED )
      Coil( "DB359_M_UNIT_02_STA_2".M_CODES_UNIT_02_STA_2.Ack_M725 )
   END_RUNG
   // the same network as SCL:
   "DB359_M_UNIT_02_STA_2".M_CODES_UNIT_02_STA_2.Ack_M725 := "DB3810_U2_F4_GRIPPER".CYL.FULL_LOW_PRESSURED;
END_REGION

REGION Network 28: M725-FIXTURE 4 GRIPPER LOW PRESSURE (READ-IN DISABLE) / M23-SWITCH ON SPINDLE FRAME BLOWING
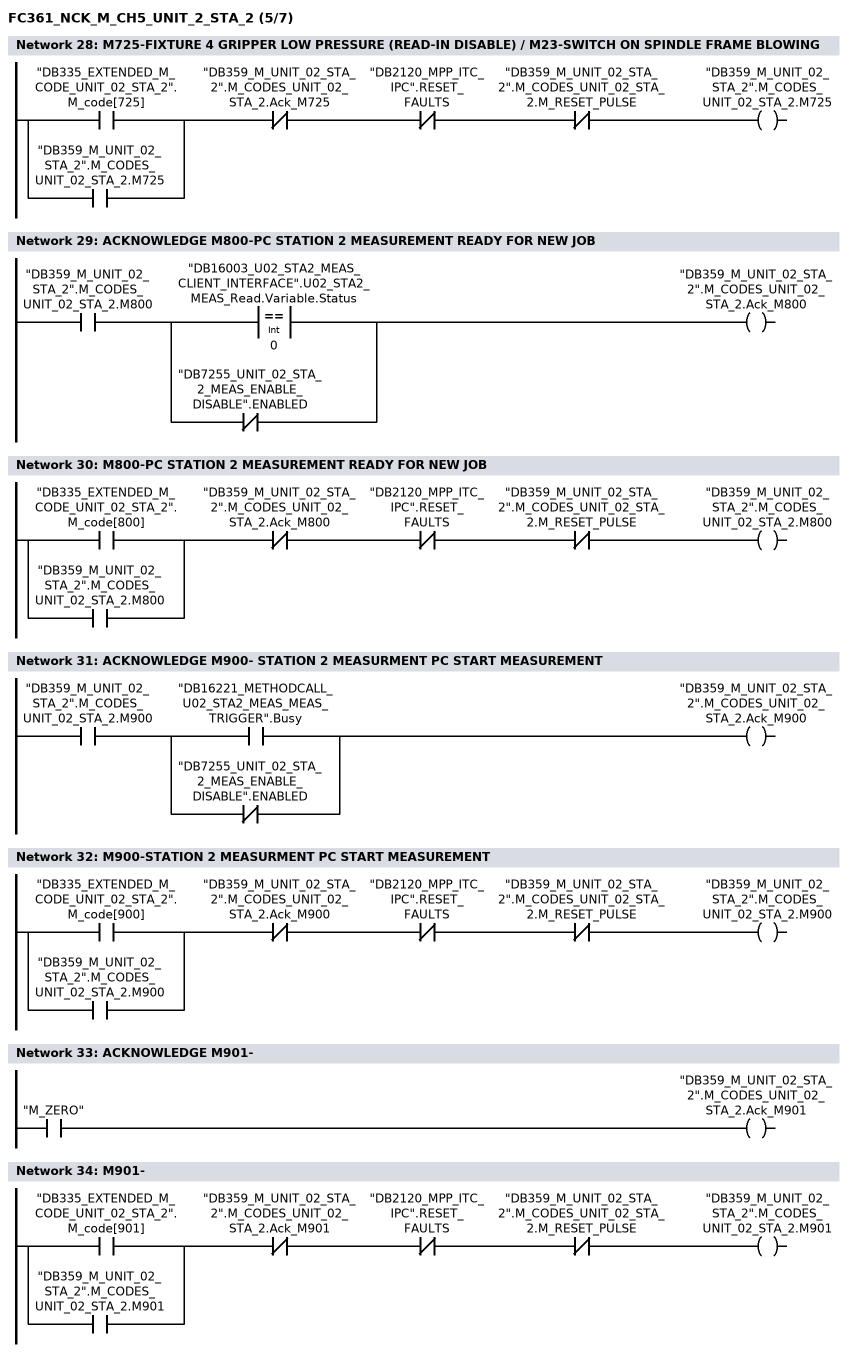
   RUNG wire#powerrail
      Contact( "DB335_EXTENDED_M_CODE_UNIT_02_STA_2".M_code[725] )
      wire#w1
      I_Contact( "DB359_M_UNIT_02_STA_2".M_CODES_UNIT_02_STA_2.Ack_M725 )
      I_Contact( "DB2120_MPP_ITC_IPC".RESET_FAULTS )
      I_Contact( "DB359_M_UNIT_02_STA_2".M_CODES_UNIT_02_STA_2.M_RESET_PULSE )
      Coil( "DB359_M_UNIT_02_STA_2".M_CODES_UNIT_02_STA_2.M725 )
   END_RUNG
   RUNG wire#powerrail
      Contact( "DB359_M_UNIT_02_STA_2".M_CODES_UNIT_02_STA_2.M725 )
   END_RUNG wire#w1
   // the same network as SCL:
   "DB359_M_UNIT_02_STA_2".M_CODES_UNIT_02_STA_2.M725 := ("DB335_EXTENDED_M_CODE_UNIT_02_STA_2".M_code[725] OR "DB359_M_UNIT_02_STA_2".M_CODES_UNIT_02_STA_2.M725) AND NOT "DB359_M_UNIT_02_STA_2".M_CODES_UNIT_02_STA_2.Ack_M725 AND NOT "DB2120_MPP_ITC_IPC".RESET_FAULTS AND NOT "DB359_M_UNIT_02_STA_2".M_CODES_UNIT_02_STA_2.M_RESET_PULSE;
END_REGION

REGION Network 29: ACKNOWLEDGE M800-PC STATION 2 MEASUREMENT READY FOR NEW JOB
   RUNG wire#powerrail
      Contact( "DB359_M_UNIT_02_STA_2".M_CODES_UNIT_02_STA_2.M800 )
      wire#w1
      { S7_Templates := "SrcType := Int" } EQ_Contact(in1 := "DB16003_U02_STA2_MEAS_CLIENT_INTERFACE".U02_STA2_MEAS_Read.Variable.Status, in2 := 0)
      wire#w2
      Coil( "DB359_M_UNIT_02_STA_2".M_CODES_UNIT_02_STA_2.Ack_M800 )
   END_RUNG
   RUNG wire#w1
      I_Contact( "DB7255_UNIT_02_STA_2_MEAS_ENABLE_DISABLE".ENABLED )
   END_RUNG wire#w2
   // the same network as SCL:
   "DB359_M_UNIT_02_STA_2".M_CODES_UNIT_02_STA_2.Ack_M800 := "DB359_M_UNIT_02_STA_2".M_CODES_UNIT_02_STA_2.M800 AND (("DB16003_U02_STA2_MEAS_CLIENT_INTERFACE".U02_STA2_MEAS_Read.Variable.Status = 0) OR NOT "DB7255_UNIT_02_STA_2_MEAS_ENABLE_DISABLE".ENABLED);
END_REGION

REGION Network 30: M800-PC STATION 2 MEASUREMENT READY FOR NEW JOB
   RUNG wire#powerrail
      Contact( "DB335_EXTENDED_M_CODE_UNIT_02_STA_2".M_code[800] )
      wire#w1
      I_Contact( "DB359_M_UNIT_02_STA_2".M_CODES_UNIT_02_STA_2.Ack_M800 )
      I_Contact( "DB2120_MPP_ITC_IPC".RESET_FAULTS )
      I_Contact( "DB359_M_UNIT_02_STA_2".M_CODES_UNIT_02_STA_2.M_RESET_PULSE )
      Coil( "DB359_M_UNIT_02_STA_2".M_CODES_UNIT_02_STA_2.M800 )
   END_RUNG
   RUNG wire#powerrail
      Contact( "DB359_M_UNIT_02_STA_2".M_CODES_UNIT_02_STA_2.M800 )
   END_RUNG wire#w1
   // the same network as SCL:
   "DB359_M_UNIT_02_STA_2".M_CODES_UNIT_02_STA_2.M800 := ("DB335_EXTENDED_M_CODE_UNIT_02_STA_2".M_code[800] OR "DB359_M_UNIT_02_STA_2".M_CODES_UNIT_02_STA_2.M800) AND NOT "DB359_M_UNIT_02_STA_2".M_CODES_UNIT_02_STA_2.Ack_M800 AND NOT "DB2120_MPP_ITC_IPC".RESET_FAULTS AND NOT "DB359_M_UNIT_02_STA_2".M_CODES_UNIT_02_STA_2.M_RESET_PULSE;
END_REGION

REGION Network 31: ACKNOWLEDGE M900- STATION 2 MEASURMENT PC START MEASUREMENT
   RUNG wire#powerrail
      Contact( "DB359_M_UNIT_02_STA_2".M_CODES_UNIT_02_STA_2.M900 )
      wire#w1
      Contact( "DB16221_METHODCALL_U02_STA2_MEAS_MEAS_TRIGGER".Busy )
      wire#w2
      Coil( "DB359_M_UNIT_02_STA_2".M_CODES_UNIT_02_STA_2.Ack_M900 )
   END_RUNG
   RUNG wire#w1
      I_Contact( "DB7255_UNIT_02_STA_2_MEAS_ENABLE_DISABLE".ENABLED )
   END_RUNG wire#w2
   // the same network as SCL:
   "DB359_M_UNIT_02_STA_2".M_CODES_UNIT_02_STA_2.Ack_M900 := "DB359_M_UNIT_02_STA_2".M_CODES_UNIT_02_STA_2.M900 AND ("DB16221_METHODCALL_U02_STA2_MEAS_MEAS_TRIGGER".Busy OR NOT "DB7255_UNIT_02_STA_2_MEAS_ENABLE_DISABLE".ENABLED);
END_REGION

REGION Network 32: M900-STATION 2 MEASURMENT PC START MEASUREMENT
   RUNG wire#powerrail
      Contact( "DB335_EXTENDED_M_CODE_UNIT_02_STA_2".M_code[900] )
      wire#w1
      I_Contact( "DB359_M_UNIT_02_STA_2".M_CODES_UNIT_02_STA_2.Ack_M900 )
      I_Contact( "DB2120_MPP_ITC_IPC".RESET_FAULTS )
      I_Contact( "DB359_M_UNIT_02_STA_2".M_CODES_UNIT_02_STA_2.M_RESET_PULSE )
      Coil( "DB359_M_UNIT_02_STA_2".M_CODES_UNIT_02_STA_2.M900 )
   END_RUNG
   RUNG wire#powerrail
      Contact( "DB359_M_UNIT_02_STA_2".M_CODES_UNIT_02_STA_2.M900 )
   END_RUNG wire#w1
   // the same network as SCL:
   "DB359_M_UNIT_02_STA_2".M_CODES_UNIT_02_STA_2.M900 := ("DB335_EXTENDED_M_CODE_UNIT_02_STA_2".M_code[900] OR "DB359_M_UNIT_02_STA_2".M_CODES_UNIT_02_STA_2.M900) AND NOT "DB359_M_UNIT_02_STA_2".M_CODES_UNIT_02_STA_2.Ack_M900 AND NOT "DB2120_MPP_ITC_IPC".RESET_FAULTS AND NOT "DB359_M_UNIT_02_STA_2".M_CODES_UNIT_02_STA_2.M_RESET_PULSE;
END_REGION

REGION Network 33: ACKNOWLEDGE M901-
   RUNG wire#powerrail
      Contact( "M_ZERO" )
      Coil( "DB359_M_UNIT_02_STA_2".M_CODES_UNIT_02_STA_2.Ack_M901 )
   END_RUNG
   // the same network as SCL:
   "DB359_M_UNIT_02_STA_2".M_CODES_UNIT_02_STA_2.Ack_M901 := "M_ZERO";
END_REGION

REGION Network 34: M901-
   RUNG wire#powerrail
      Contact( "DB335_EXTENDED_M_CODE_UNIT_02_STA_2".M_code[901] )
      wire#w1
      I_Contact( "DB359_M_UNIT_02_STA_2".M_CODES_UNIT_02_STA_2.Ack_M901 )
      I_Contact( "DB2120_MPP_ITC_IPC".RESET_FAULTS )
      I_Contact( "DB359_M_UNIT_02_STA_2".M_CODES_UNIT_02_STA_2.M_RESET_PULSE )
      Coil( "DB359_M_UNIT_02_STA_2".M_CODES_UNIT_02_STA_2.M901 )
   END_RUNG
   RUNG wire#powerrail
      Contact( "DB359_M_UNIT_02_STA_2".M_CODES_UNIT_02_STA_2.M901 )
   END_RUNG wire#w1
   // the same network as SCL:
   "DB359_M_UNIT_02_STA_2".M_CODES_UNIT_02_STA_2.M901 := ("DB335_EXTENDED_M_CODE_UNIT_02_STA_2".M_code[901] OR "DB359_M_UNIT_02_STA_2".M_CODES_UNIT_02_STA_2.M901) AND NOT "DB359_M_UNIT_02_STA_2".M_CODES_UNIT_02_STA_2.Ack_M901 AND NOT "DB2120_MPP_ITC_IPC".RESET_FAULTS AND NOT "DB359_M_UNIT_02_STA_2".M_CODES_UNIT_02_STA_2.M_RESET_PULSE;
END_REGION

REGION Network 35: ACKNOWLEDGE M902-
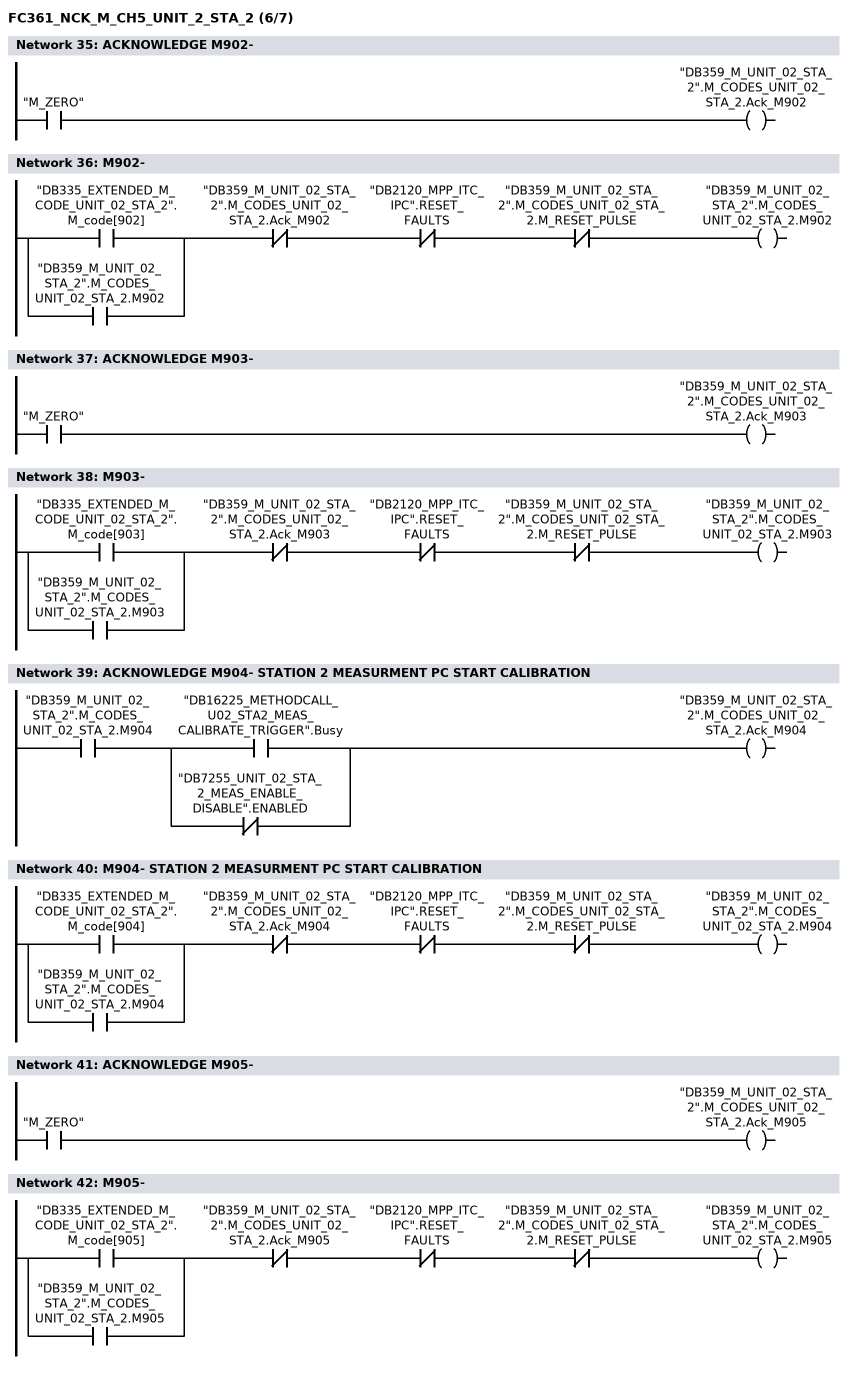
   RUNG wire#powerrail
      Contact( "M_ZERO" )
      Coil( "DB359_M_UNIT_02_STA_2".M_CODES_UNIT_02_STA_2.Ack_M902 )
   END_RUNG
   // the same network as SCL:
   "DB359_M_UNIT_02_STA_2".M_CODES_UNIT_02_STA_2.Ack_M902 := "M_ZERO";
END_REGION

REGION Network 36: M902-
   RUNG wire#powerrail
      Contact( "DB335_EXTENDED_M_CODE_UNIT_02_STA_2".M_code[902] )
      wire#w1
      I_Contact( "DB359_M_UNIT_02_STA_2".M_CODES_UNIT_02_STA_2.Ack_M902 )
      I_Contact( "DB2120_MPP_ITC_IPC".RESET_FAULTS )
      I_Contact( "DB359_M_UNIT_02_STA_2".M_CODES_UNIT_02_STA_2.M_RESET_PULSE )
      Coil( "DB359_M_UNIT_02_STA_2".M_CODES_UNIT_02_STA_2.M902 )
   END_RUNG
   RUNG wire#powerrail
      Contact( "DB359_M_UNIT_02_STA_2".M_CODES_UNIT_02_STA_2.M902 )
   END_RUNG wire#w1
   // the same network as SCL:
   "DB359_M_UNIT_02_STA_2".M_CODES_UNIT_02_STA_2.M902 := ("DB335_EXTENDED_M_CODE_UNIT_02_STA_2".M_code[902] OR "DB359_M_UNIT_02_STA_2".M_CODES_UNIT_02_STA_2.M902) AND NOT "DB359_M_UNIT_02_STA_2".M_CODES_UNIT_02_STA_2.Ack_M902 AND NOT "DB2120_MPP_ITC_IPC".RESET_FAULTS AND NOT "DB359_M_UNIT_02_STA_2".M_CODES_UNIT_02_STA_2.M_RESET_PULSE;
END_REGION

REGION Network 37: ACKNOWLEDGE M903-
   RUNG wire#powerrail
      Contact( "M_ZERO" )
      Coil( "DB359_M_UNIT_02_STA_2".M_CODES_UNIT_02_STA_2.Ack_M903 )
   END_RUNG
   // the same network as SCL:
   "DB359_M_UNIT_02_STA_2".M_CODES_UNIT_02_STA_2.Ack_M903 := "M_ZERO";
END_REGION

REGION Network 38: M903-
   RUNG wire#powerrail
      Contact( "DB335_EXTENDED_M_CODE_UNIT_02_STA_2".M_code[903] )
      wire#w1
      I_Contact( "DB359_M_UNIT_02_STA_2".M_CODES_UNIT_02_STA_2.Ack_M903 )
      I_Contact( "DB2120_MPP_ITC_IPC".RESET_FAULTS )
      I_Contact( "DB359_M_UNIT_02_STA_2".M_CODES_UNIT_02_STA_2.M_RESET_PULSE )
      Coil( "DB359_M_UNIT_02_STA_2".M_CODES_UNIT_02_STA_2.M903 )
   END_RUNG
   RUNG wire#powerrail
      Contact( "DB359_M_UNIT_02_STA_2".M_CODES_UNIT_02_STA_2.M903 )
   END_RUNG wire#w1
   // the same network as SCL:
   "DB359_M_UNIT_02_STA_2".M_CODES_UNIT_02_STA_2.M903 := ("DB335_EXTENDED_M_CODE_UNIT_02_STA_2".M_code[903] OR "DB359_M_UNIT_02_STA_2".M_CODES_UNIT_02_STA_2.M903) AND NOT "DB359_M_UNIT_02_STA_2".M_CODES_UNIT_02_STA_2.Ack_M903 AND NOT "DB2120_MPP_ITC_IPC".RESET_FAULTS AND NOT "DB359_M_UNIT_02_STA_2".M_CODES_UNIT_02_STA_2.M_RESET_PULSE;
END_REGION

REGION Network 39: ACKNOWLEDGE M904- STATION 2 MEASURMENT PC START CALIBRATION
   RUNG wire#powerrail
      Contact( "DB359_M_UNIT_02_STA_2".M_CODES_UNIT_02_STA_2.M904 )
      wire#w1
      Contact( "DB16225_METHODCALL_U02_STA2_MEAS_CALIBRATE_TRIGGER".Busy )
      wire#w2
      Coil( "DB359_M_UNIT_02_STA_2".M_CODES_UNIT_02_STA_2.Ack_M904 )
   END_RUNG
   RUNG wire#w1
      I_Contact( "DB7255_UNIT_02_STA_2_MEAS_ENABLE_DISABLE".ENABLED )
   END_RUNG wire#w2
   // the same network as SCL:
   "DB359_M_UNIT_02_STA_2".M_CODES_UNIT_02_STA_2.Ack_M904 := "DB359_M_UNIT_02_STA_2".M_CODES_UNIT_02_STA_2.M904 AND ("DB16225_METHODCALL_U02_STA2_MEAS_CALIBRATE_TRIGGER".Busy OR NOT "DB7255_UNIT_02_STA_2_MEAS_ENABLE_DISABLE".ENABLED);
END_REGION

REGION Network 40: M904- STATION 2 MEASURMENT PC START CALIBRATION
   RUNG wire#powerrail
      Contact( "DB335_EXTENDED_M_CODE_UNIT_02_STA_2".M_code[904] )
      wire#w1
      I_Contact( "DB359_M_UNIT_02_STA_2".M_CODES_UNIT_02_STA_2.Ack_M904 )
      I_Contact( "DB2120_MPP_ITC_IPC".RESET_FAULTS )
      I_Contact( "DB359_M_UNIT_02_STA_2".M_CODES_UNIT_02_STA_2.M_RESET_PULSE )
      Coil( "DB359_M_UNIT_02_STA_2".M_CODES_UNIT_02_STA_2.M904 )
   END_RUNG
   RUNG wire#powerrail
      Contact( "DB359_M_UNIT_02_STA_2".M_CODES_UNIT_02_STA_2.M904 )
   END_RUNG wire#w1
   // the same network as SCL:
   "DB359_M_UNIT_02_STA_2".M_CODES_UNIT_02_STA_2.M904 := ("DB335_EXTENDED_M_CODE_UNIT_02_STA_2".M_code[904] OR "DB359_M_UNIT_02_STA_2".M_CODES_UNIT_02_STA_2.M904) AND NOT "DB359_M_UNIT_02_STA_2".M_CODES_UNIT_02_STA_2.Ack_M904 AND NOT "DB2120_MPP_ITC_IPC".RESET_FAULTS AND NOT "DB359_M_UNIT_02_STA_2".M_CODES_UNIT_02_STA_2.M_RESET_PULSE;
END_REGION

REGION Network 41: ACKNOWLEDGE M905-
   RUNG wire#powerrail
      Contact( "M_ZERO" )
      Coil( "DB359_M_UNIT_02_STA_2".M_CODES_UNIT_02_STA_2.Ack_M905 )
   END_RUNG
   // the same network as SCL:
   "DB359_M_UNIT_02_STA_2".M_CODES_UNIT_02_STA_2.Ack_M905 := "M_ZERO";
END_REGION

REGION Network 42: M905-
   RUNG wire#powerrail
      Contact( "DB335_EXTENDED_M_CODE_UNIT_02_STA_2".M_code[905] )
      wire#w1
      I_Contact( "DB359_M_UNIT_02_STA_2".M_CODES_UNIT_02_STA_2.Ack_M905 )
      I_Contact( "DB2120_MPP_ITC_IPC".RESET_FAULTS )
      I_Contact( "DB359_M_UNIT_02_STA_2".M_CODES_UNIT_02_STA_2.M_RESET_PULSE )
      Coil( "DB359_M_UNIT_02_STA_2".M_CODES_UNIT_02_STA_2.M905 )
   END_RUNG
   RUNG wire#powerrail
      Contact( "DB359_M_UNIT_02_STA_2".M_CODES_UNIT_02_STA_2.M905 )
   END_RUNG wire#w1
   // the same network as SCL:
   "DB359_M_UNIT_02_STA_2".M_CODES_UNIT_02_STA_2.M905 := ("DB335_EXTENDED_M_CODE_UNIT_02_STA_2".M_code[905] OR "DB359_M_UNIT_02_STA_2".M_CODES_UNIT_02_STA_2.M905) AND NOT "DB359_M_UNIT_02_STA_2".M_CODES_UNIT_02_STA_2.Ack_M905 AND NOT "DB2120_MPP_ITC_IPC".RESET_FAULTS AND NOT "DB359_M_UNIT_02_STA_2".M_CODES_UNIT_02_STA_2.M_RESET_PULSE;
END_REGION

REGION Network 43: READ-IN DISABLE / Read-in disable
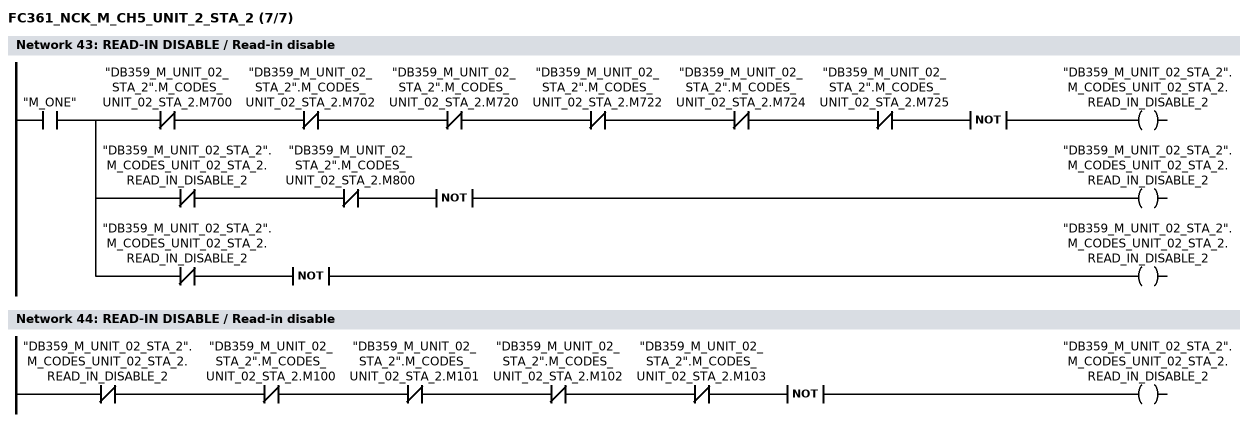
   RUNG wire#powerrail
      Contact( "M_ONE" )
      wire#w1
      I_Contact( "DB359_M_UNIT_02_STA_2".M_CODES_UNIT_02_STA_2.M700 )
      I_Contact( "DB359_M_UNIT_02_STA_2".M_CODES_UNIT_02_STA_2.M702 )
      I_Contact( "DB359_M_UNIT_02_STA_2".M_CODES_UNIT_02_STA_2.M720 )
      I_Contact( "DB359_M_UNIT_02_STA_2".M_CODES_UNIT_02_STA_2.M722 )
      I_Contact( "DB359_M_UNIT_02_STA_2".M_CODES_UNIT_02_STA_2.M724 )
      I_Contact( "DB359_M_UNIT_02_STA_2".M_CODES_UNIT_02_STA_2.M725 )
      Not()
      Coil( "DB359_M_UNIT_02_STA_2".M_CODES_UNIT_02_STA_2.READ_IN_DISABLE_2 )
   END_RUNG
   RUNG wire#w1
      I_Contact( "DB359_M_UNIT_02_STA_2".M_CODES_UNIT_02_STA_2.READ_IN_DISABLE_2 )
      I_Contact( "DB359_M_UNIT_02_STA_2".M_CODES_UNIT_02_STA_2.M800 )
      Not()
      Coil( "DB359_M_UNIT_02_STA_2".M_CODES_UNIT_02_STA_2.READ_IN_DISABLE_2 )
   END_RUNG
   RUNG wire#w1
      I_Contact( "DB359_M_UNIT_02_STA_2".M_CODES_UNIT_02_STA_2.READ_IN_DISABLE_2 )
      Not()
      Coil( "DB359_M_UNIT_02_STA_2".M_CODES_UNIT_02_STA_2.READ_IN_DISABLE_2 )
   END_RUNG
   // the same network as SCL:
   "DB359_M_UNIT_02_STA_2".M_CODES_UNIT_02_STA_2.READ_IN_DISABLE_2 := NOT ("M_ONE" AND NOT "DB359_M_UNIT_02_STA_2".M_CODES_UNIT_02_STA_2.M700 AND NOT "DB359_M_UNIT_02_STA_2".M_CODES_UNIT_02_STA_2.M702 AND NOT "DB359_M_UNIT_02_STA_2".M_CODES_UNIT_02_STA_2.M720 AND NOT "DB359_M_UNIT_02_STA_2".M_CODES_UNIT_02_STA_2.M722 AND NOT "DB359_M_UNIT_02_STA_2".M_CODES_UNIT_02_STA_2.M724 AND NOT "DB359_M_UNIT_02_STA_2".M_CODES_UNIT_02_STA_2.M725);
   "DB359_M_UNIT_02_STA_2".M_CODES_UNIT_02_STA_2.READ_IN_DISABLE_2 := NOT ("M_ONE" AND NOT "DB359_M_UNIT_02_STA_2".M_CODES_UNIT_02_STA_2.READ_IN_DISABLE_2 AND NOT "DB359_M_UNIT_02_STA_2".M_CODES_UNIT_02_STA_2.M800);
   "DB359_M_UNIT_02_STA_2".M_CODES_UNIT_02_STA_2.READ_IN_DISABLE_2 := NOT ("M_ONE" AND NOT "DB359_M_UNIT_02_STA_2".M_CODES_UNIT_02_STA_2.READ_IN_DISABLE_2);
END_REGION

REGION Network 44: READ-IN DISABLE / Read-in disable
   RUNG wire#powerrail
      I_Contact( "DB359_M_UNIT_02_STA_2".M_CODES_UNIT_02_STA_2.READ_IN_DISABLE_2 )
      I_Contact( "DB359_M_UNIT_02_STA_2".M_CODES_UNIT_02_STA_2.M100 )
      I_Contact( "DB359_M_UNIT_02_STA_2".M_CODES_UNIT_02_STA_2.M101 )
      I_Contact( "DB359_M_UNIT_02_STA_2".M_CODES_UNIT_02_STA_2.M102 )
      I_Contact( "DB359_M_UNIT_02_STA_2".M_CODES_UNIT_02_STA_2.M103 )
      Not()
      Coil( "DB359_M_UNIT_02_STA_2".M_CODES_UNIT_02_STA_2.READ_IN_DISABLE_2 )
   END_RUNG
   // the same network as SCL:
   "DB359_M_UNIT_02_STA_2".M_CODES_UNIT_02_STA_2.READ_IN_DISABLE_2 := NOT (NOT "DB359_M_UNIT_02_STA_2".M_CODES_UNIT_02_STA_2.READ_IN_DISABLE_2 AND NOT "DB359_M_UNIT_02_STA_2".M_CODES_UNIT_02_STA_2.M100 AND NOT "DB359_M_UNIT_02_STA_2".M_CODES_UNIT_02_STA_2.M101 AND NOT "DB359_M_UNIT_02_STA_2".M_CODES_UNIT_02_STA_2.M102 AND NOT "DB359_M_UNIT_02_STA_2".M_CODES_UNIT_02_STA_2.M103);
END_REGION
END_FUNCTION
